FUNCTION_BLOCK ADD_3 (* Calculate arithmetical sum of magnitude inputs (generic FB) *)
  {SET_ATTRIBUTE(eclipse4diac::core::GenericClassName, 'GEN_ADD')}
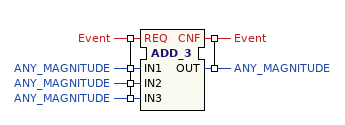
  EVENT_INPUT
    REQ WITH IN1, IN2, IN3; (* Normal Execution Request *)
  END_EVENT
  EVENT_OUTPUT
    CNF WITH OUT; (* Execution Confirmation *)
  END_EVENT
  VAR_INPUT
    IN1 : ANY_MAGNITUDE; (* ADD input 1 *)
    IN2 : ANY_MAGNITUDE; (* ADD input 2 *)
    IN3 : ANY_MAGNITUDE; (* ADD input 3 *)
  END_VAR
  VAR_OUTPUT
    OUT : ANY_MAGNITUDE; (* ADD result *)
  END_VAR
END_FUNCTION_BLOCK
